// TIA Portal V16 export
// export: Created 2024-04-23T10:19:31.9118753Z, ExportSetting WithDefaults, DisplayName Totally Integrated Automation Portal, DisplayVersion V16 Update 5, DisplayName TIA Portal Version Control Interface, DisplayVersion V16 Update 2, DisplayName TIA Portal Openness, DisplayVersion V16 Update 5, DisplayName TIA Portal Teamcenter Gateway, DisplayVersion V16, DisplayName SINAMICS Startdrive Advanced, DisplayVersion V16, DisplayName SINAMICS Startdrive G130, G150, S120, S150, SINAMICS MV, S210, DisplayVersion V16, DisplayName SINAMICS Startdrive G110M, G120, G120C, G120D, G120P, DisplayVersion V16, DisplayName STEP 7 Professional, DisplayVersion V16 Update 5, DisplayName STEP 7 Safety, DisplayVersion V16, DisplayName WinCC UA Professional, DisplayVersion V16 Update 5
FUNCTION_BLOCK "Calculo de Seno"   // FB1, LAD
{ S7_Optimized_Access := 'TRUE' }
VERSION : 0.1
// stored: AutoNumber true, IsIECCheckEnabled false, IsRetainMemResEnabled false, MemoryReserve 100, SetENOAutomatically false, UDAEnableTagReadback false
   VAR_OUTPUT
      SenOUT : Real;
   END_VAR
   VAR_IN_OUT
      SenIN : Real;
   END_VAR
   VAR
      Pulso1ms : Bool;
      AuxPulso1ms : Bool;
      AuxFlancoPulso4ms : Bool;
      Flanco4ms { ExternalAccessible := 'False'; ExternalVisible := 'False'; ExternalWritable := 'False'} : Bool;
   END_VAR
   VAR_TEMP
      SenAUX : Real;
      "SenIN-Radianes" : Real;
   END_VAR
   VAR CONSTANT
      PI : Real := 3.1416;
   END_VAR
BEGIN

REGION Network 1
   // Pasar de grados a radianes
END_REGION

REGION Network 2 (SCL)
   "Timer1".TON(IN := #AuxPulso1ms,
                PT := T#10ms,
                Q => #Pulso1ms);

   "Timer2".TOF(IN := NOT #Pulso1ms,
                PT := T#10ms,
                Q => #AuxPulso1ms);

   #Flanco4ms := NOT #Flanco4ms AND #Pulso1ms;

   IF #Pulso1ms THEN
       #SenIN := #SenIN + 1;
   END_IF;

   IF #SenIN >= 360.0 THEN
       #SenIN := 0.0;
   END_IF;

   #"SenIN-Radianes" := (#SenIN * #PI) / 180.0;

   #SenOUT := SIN(#"SenIN-Radianes");
END_REGION
END_FUNCTION_BLOCK
